(* PLC project Generated.project, CODESYS CODESYS V3.5 SP19 Patch 1 *)
(* stored: creationDateTime 2026-09-06T13:00:42.565323, modificationDateTime 2026-09-06T13:00:42.565323 *)

(* ═══════════════════════════════════════════════════════════════ 🎮 ST_SyncCmd — Commandes IHM pour la synchronisation M1/M2 ═══════════════════════════════════════════════════════════════ *)
TYPE ST_SyncCmd : STRUCT
  SelSyncEnable : BOOL := TRUE;  (* ☑️ coché = synchro voulue (MAINT_N1/N2) *)
END_STRUCT;
END_TYPE
